FUNCTION_BLOCK DATA_ACUM
  {SET_ATTRIBUTE(OpcUa, SERVICE)}
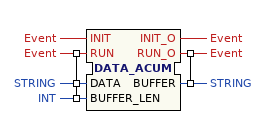
  EVENT_INPUT
    INIT;
    RUN WITH DATA, BUFFER_LEN;
  END_EVENT
  EVENT_OUTPUT
    INIT_O;
    RUN_O WITH BUFFER;
  END_EVENT
  VAR_INPUT
    DATA : STRING;
    BUFFER_LEN : INT;
  END_VAR
  VAR_OUTPUT
    BUFFER : STRING;
  END_VAR
END_FUNCTION_BLOCK
